TYPE E_HomeSwitchTypeClass:
(
    eNoSwitch := 0, //no physical switch for homing present
    eHomeSwitchPresent := 1, //dedicated homing switch present
    eUseBwdLimit := 2, //Bwd limit switch is used as a homing switch
    eUseFwdLimit := 3 //Fwd limit switch is used as a homing switch
) := eNoSwitch;
END_TYPE

(* stored: Version 1.1.0.1, ProductVersion 3.1.4024.11
   DUT E_HomeSwitchTypeClass: Id {efe4c9b6-f0fb-4dcd-aeb8-a35b3f20f344} *)
